# EPICS IOC start-up script: motorApp/iocsh/allstop.iocsh
# ### allstop.iocsh ###

#- ###################################################
#- PREFIX           - IOC Prefix
#- MOTOR            - Location of motor module
#- ###################################################

#- Allstop, alldone
dbLoadRecords("$(MOTOR)/db/motorUtil.db", "P=$(PREFIX)")
doAfterIocInit("motorUtilInit('$(PREFIX)')")
